PROGRAM MAIN
VAR

END_VAR

Systemzeit();
Blinker();
//Line_Chart_array();

//LineChart();
//TOF_Beispiel();

alle_5sekunden();

END_PROGRAM

(* stored: Version 1.1.0.1
   POU MAIN: Id {d4e7d423-fa3e-4ab1-8f91-d0cc7021abc2}, SpecialFunc None *)
